# EPICS substitutions: tpmacApp/Db/pmac_asyn_motor.substitutions
file "db/pmac_asyn_motor.db"
{
pattern
{SYS,            DEV,               MOTOR,  SPORT,  ADDR,  DESC,             DTYP        PREC,  EGU}
{"XF:03IDB-OP",  "{BPM:7-Ax:Y}",    "M0",   "P0",   1,     "Y Translation",  asynMotor,  9,     "mm"}
}
